{attribute 'qualified_only'}
{attribute 'strict'}
TYPE E_EventType :
(
	Alarm :=0,
	Message :=1
);
END_TYPE

(* stored: Version 1.1.0.1, ProductVersion 3.1.4024.12
   DUT E_EventType: Id {9673939b-76fd-4c81-80cd-8291a53c722e} *)
